(*

short summary
==================
This class tests all methods of xint assertions
with various combinations of inputs and checks expected 
outputs are satisfied or not

.. <legal notes>

legal notes
=================
| SPDX-FileCopyrightText: © 2022 ekvip automation GmbH <info@ekvip.de>
| SPDX-License-Identifier: Apache-2.0
| For details check: Apache-2.0_

.. _Apache-2.0: https://www.apache.org/licenses/LICENSE-2.0

.. </legal notes>

methods and properties
======================

*)

FUNCTION_BLOCK XintAssertionTests EXTENDS AbstractAssertorTest
VAR_INPUT
END_VAR
VAR CONSTANT
	(* prefix to unify the test names *)
	TEST_NAME_PREFIX	:Tc2_System.T_MaxString := 'assert.integer.signed.x.';
	(* number of the lsb *)
	FIRST_BIT				:USINT := 0;
	(* number of the msb *)
	LAST_BIT				:USINT := ((SIZEOF(__XINT)*8)-1);
	(* since we don't know the lenght of __XINT we need it to initialize ``MULTIPLICAND`` *)
	{attribute 'hide'}
	INIT_VALUE_MULTIPLICAND	:__XWORD := 16#1111_1111;
	(* multiplicand for the ``multiplier`` *)
	MULTIPLICAND			:__XINT := (ROR(INIT_VALUE_MULTIPLICAND, 32) OR INIT_VALUE_MULTIPLICAND);
	(* first of all multipliers the test iterates *)
	FIRST_MULTIPLIER		:__XINT := 0;
	(* first of all multipliers the test iterates *)
	LAST_MULTIPLIER			:__XINT := 15;
	(* just the value zero *)
	ZERO					:__XINT := 0;
	(* just the lsb is set, it's just the value one *)
	LSB_ONLY				:__XINT := 1;
	(* all bits are set *)
	ALL_BITS_SET			:__XINT := -1;
	(* the msb is set only *)
	MINIMUM_VALUE			:__XINT := ROR(LSB_ONLY,1);
	(* 
	since we don't know the lenght of __XINT 
	we need it to initialize ``MAXIMUM_VALUE``.
	SHR is not working with __XINT
	*)
	{attribute 'hide'}
	BINARY_MINUS_ONE		:__XWORD := ALL_BITS_SET;
	(* the msb is unset only *)
	MAXIMUM_VALUE			:__XINT := SHR(BINARY_MINUS_ONE,1);
END_VAR

THIS^.runValueIsEqualToTests();
THIS^.runValueIsEvenTests();
THIS^.runValueIsGreaterTests();
THIS^.runValueIsInRangeOfTests();
THIS^.runValueIsLessThanTests();
THIS^.runValueIsMaxTests();
THIS^.runValueIsMinTests();
THIS^.runValueIsNegativeTests();
THIS^.runValueIsNotEqualToTests();
THIS^.runValueIsOddTests();
THIS^.runValueIsPositiveTests();

(*

short summary
==================
This test method is a helper function to create a unified test name

.. <legal notes>

legal notes
=================
| SPDX-FileCopyrightText: © 2022 ekvip automation GmbH <info@ekvip.de>
| SPDX-License-Identifier: Apache-2.0
| For details check: Apache-2.0_

.. _Apache-2.0: https://www.apache.org/licenses/LICENSE-2.0

.. </legal notes>

parameters
==========

*)

METHOD PROTECTED getTestNameFor :Tc2_System.T_MaxString
VAR_INPUT
	(* name of the method to test, to create a unified test name *)
	nameOfMethodToTest	:Tc2_System.T_MaxString;
END_VAR
getTestNameFor := Tc2_Standard.CONCAT(THIS^.TEST_NAME_PREFIX, nameOfMethodToTest);
END_METHOD

(*

short summary
==================
This test method tests ``assert.integer.signed.x.valueIsEqualTo``
method of CNM_AssertionInterfaceLib library with various inputs

.. <legal notes>

legal notes
=================
| SPDX-FileCopyrightText: © 2022 ekvip automation GmbH <info@ekvip.de>
| SPDX-License-Identifier: Apache-2.0
| For details check: Apache-2.0_

.. _Apache-2.0: https://www.apache.org/licenses/LICENSE-2.0

.. </legal notes>

*)

METHOD runValueIsEqualToTests
RETURN (NOT TcUnit.TEST_ORDERED(THIS^.getTestNameFor('valueIsEqualTo')));

THIS^.testValueIsEqualTo(
	valueToTest := THIS^.ZERO,
	expected := THIS^.ALL_BITS_SET
);
THIS^.testValueIsEqualTo(
	valueToTest := THIS^.ZERO,
	expected := THIS^.ZERO
);
THIS^.testValueIsEqualTo(
	valueToTest := THIS^.ALL_BITS_SET,
	expected := THIS^.ALL_BITS_SET
);
THIS^.testValueIsEqualTo(
	valueToTest := THIS^.ALL_BITS_SET,
	expected := THIS^.ZERO
);
THIS^.testValueIsEqualTo(
	valueToTest := THIS^.LSB_ONLY,
	expected := THIS^.LSB_ONLY
);
THIS^.testValueIsEqualTo(
	valueToTest := THIS^.LSB_ONLY,
	expected := THIS^.MINIMUM_VALUE
);
THIS^.testValueIsEqualTo(
	valueToTest := THIS^.MINIMUM_VALUE,
	expected := THIS^.MINIMUM_VALUE
);
THIS^.testValueIsEqualTo(
	valueToTest := THIS^.MINIMUM_VALUE,
	expected := THIS^.LSB_ONLY
);
THIS^.testValueIsEqualTo(
	valueToTest := THIS^.MINIMUM_VALUE,
	expected := THIS^.MAXIMUM_VALUE
);

TcUnit.TEST_FINISHED();
END_METHOD

(*

short summary
==================
This test method tests ``assert.integer.signed.x.valueIsEven``
of CNM_AssertionInterfaceLib library with various inputs

.. <legal notes>

legal notes
=================
| SPDX-FileCopyrightText: © 2022 ekvip automation GmbH <info@ekvip.de>
| SPDX-License-Identifier: Apache-2.0
| For details check: Apache-2.0_

.. _Apache-2.0: https://www.apache.org/licenses/LICENSE-2.0

.. </legal notes>

*)

METHOD runValueIsEvenTests
VAR
	(* it's just part of the test data *)
	valueToTest	:__XINT;
	(* multiplier to get various bit patterns *)
	multiplier	:__XINT;
END_VAR
RETURN (NOT TcUnit.TEST_ORDERED(THIS^.getTestNameFor('valueIsEven')));

FOR multiplier := THIS^.FIRST_MULTIPLIER TO THIS^.LAST_MULTIPLIER DO
	valueToTest := (THIS^.MULTIPLICAND * multiplier);
	THIS^.testValueIsEven(
		valueToTest := valueToTest
	);
END_FOR

TcUnit.TEST_FINISHED();
END_METHOD

(*

short summary
==================
This test method tests ``assert.integer.signed.x.valueIsGreaterThan``
method of CNM_AssertionInterfaceLib library with various inputs

.. <legal notes>

legal notes
=================
| SPDX-FileCopyrightText: © 2022 ekvip automation GmbH <info@ekvip.de>
| SPDX-License-Identifier: Apache-2.0
| For details check: Apache-2.0_

.. _Apache-2.0: https://www.apache.org/licenses/LICENSE-2.0

.. </legal notes>

*)

METHOD runValueIsGreaterTests
RETURN (NOT TcUnit.TEST_ORDERED(THIS^.getTestNameFor('valueIsGreaterThan')));

THIS^.testValueIsGreater(
	valueToTest := THIS^.ZERO,
	less := THIS^.ALL_BITS_SET
);
THIS^.testValueIsGreater(
	valueToTest := THIS^.ZERO,
	less := THIS^.ZERO
);
THIS^.testValueIsGreater(
	valueToTest := THIS^.ALL_BITS_SET,
	less := THIS^.ALL_BITS_SET
);
THIS^.testValueIsGreater(
	valueToTest := THIS^.ALL_BITS_SET,
	less := THIS^.ZERO
);
THIS^.testValueIsGreater(
	valueToTest := THIS^.LSB_ONLY,
	less := THIS^.LSB_ONLY
);
THIS^.testValueIsGreater(
	valueToTest := THIS^.LSB_ONLY,
	less := THIS^.ZERO
);
THIS^.testValueIsGreater(
	valueToTest := THIS^.LSB_ONLY,
	less := (THIS^.LSB_ONLY+THIS^.LSB_ONLY)
);
THIS^.testValueIsGreater(
	valueToTest := THIS^.MINIMUM_VALUE,
	less := THIS^.MINIMUM_VALUE
);
THIS^.testValueIsGreater(
	valueToTest := THIS^.MINIMUM_VALUE,
	less := THIS^.ALL_BITS_SET
);
THIS^.testValueIsGreater(
	valueToTest := THIS^.MINIMUM_VALUE,
	less := THIS^.MAXIMUM_VALUE
);
THIS^.testValueIsGreater(
	valueToTest := THIS^.MAXIMUM_VALUE,
	less := THIS^.MINIMUM_VALUE
);

TcUnit.TEST_FINISHED();
END_METHOD

(*

short summary
==================
This test method tests ``assert.integer.signed.x.valueIsInRangeOf``
method of CNM_AssertionInterfaceLib library with various inputs

.. <legal notes>

legal notes
=================
| SPDX-FileCopyrightText: © 2022 ekvip automation GmbH <info@ekvip.de>
| SPDX-License-Identifier: Apache-2.0
| For details check: Apache-2.0_

.. _Apache-2.0: https://www.apache.org/licenses/LICENSE-2.0

.. </legal notes>

*)

METHOD runValueIsInRangeOfTests
RETURN (NOT TcUnit.TEST_ORDERED(THIS^.getTestNameFor('valueIsInRangeOf')));

THIS^.testValueIsInRangeOf(
	lower := THIS^.ZERO,
	valueToTest := THIS^.LSB_ONLY,
	upper := THIS^.ALL_BITS_SET
);
THIS^.testValueIsInRangeOf(
	lower := THIS^.ZERO,
	valueToTest := THIS^.ZERO,
	upper := THIS^.ZERO
);
THIS^.testValueIsInRangeOf(
	lower := THIS^.ALL_BITS_SET,
	valueToTest := THIS^.ALL_BITS_SET,
	upper := THIS^.ALL_BITS_SET
);
THIS^.testValueIsInRangeOf(
	lower := THIS^.ALL_BITS_SET,
	valueToTest := THIS^.LSB_ONLY,
	upper := THIS^.ZERO
);
THIS^.testValueIsInRangeOf(
	lower := THIS^.ALL_BITS_SET,
	valueToTest := THIS^.ZERO,
	upper := THIS^.ZERO
);
THIS^.testValueIsInRangeOf(
	lower := THIS^.MAXIMUM_VALUE,
	valueToTest := THIS^.ZERO,
	upper := THIS^.MINIMUM_VALUE
);
THIS^.testValueIsInRangeOf(
	lower := THIS^.MINIMUM_VALUE,
	valueToTest := THIS^.ZERO,
	upper := THIS^.MAXIMUM_VALUE
);
THIS^.testValueIsInRangeOf(
	lower := THIS^.MAXIMUM_VALUE,
	valueToTest := THIS^.MINIMUM_VALUE,
	upper := THIS^.MINIMUM_VALUE
);
THIS^.testValueIsInRangeOf(
	lower := THIS^.MINIMUM_VALUE,
	valueToTest := THIS^.MAXIMUM_VALUE,
	upper := THIS^.MAXIMUM_VALUE
);
THIS^.testValueIsInRangeOf(
	lower := THIS^.MINIMUM_VALUE,
	valueToTest := THIS^.MINIMUM_VALUE,
	upper := THIS^.MAXIMUM_VALUE
);

TEST_FINISHED();
END_METHOD

(*

short summary
==================
This test method tests ``assert.integer.signed.x.valueIsLessThan``
method of CNM_AssertionInterfaceLib library with various inputs

.. <legal notes>

legal notes
=================
| SPDX-FileCopyrightText: © 2022 ekvip automation GmbH <info@ekvip.de>
| SPDX-License-Identifier: Apache-2.0
| For details check: Apache-2.0_

.. _Apache-2.0: https://www.apache.org/licenses/LICENSE-2.0

.. </legal notes>

*)

METHOD runValueIsLessThanTests
RETURN (NOT TcUnit.TEST_ORDERED(THIS^.getTestNameFor('valueIsLessThan')));

THIS^.testValueIsLessThan(
	valueToTest := THIS^.ZERO,
	greater := THIS^.ALL_BITS_SET
);
THIS^.testValueIsLessThan(
	valueToTest := THIS^.ZERO,
	greater := THIS^.ZERO
);
THIS^.testValueIsLessThan(
	valueToTest := THIS^.ALL_BITS_SET,
	greater := THIS^.ALL_BITS_SET
);
THIS^.testValueIsLessThan(
	valueToTest := THIS^.ALL_BITS_SET,
	greater := THIS^.ZERO
);
THIS^.testValueIsLessThan(
	valueToTest := THIS^.LSB_ONLY,
	greater := THIS^.LSB_ONLY
);
THIS^.testValueIsLessThan(
	valueToTest := THIS^.LSB_ONLY,
	greater := THIS^.ZERO
);
THIS^.testValueIsLessThan(
	valueToTest := THIS^.MINIMUM_VALUE,
	greater := (THIS^.MINIMUM_VALUE+THIS^.LSB_ONLY)
);
THIS^.testValueIsLessThan(
	valueToTest := THIS^.MINIMUM_VALUE,
	greater := THIS^.MINIMUM_VALUE
);
THIS^.testValueIsLessThan(
	valueToTest := THIS^.MINIMUM_VALUE,
	greater := THIS^.ALL_BITS_SET
);
THIS^.testValueIsLessThan(
	valueToTest := THIS^.MINIMUM_VALUE,
	greater := THIS^.MAXIMUM_VALUE
);
THIS^.testValueIsLessThan(
	valueToTest := THIS^.MAXIMUM_VALUE,
	greater := THIS^.MINIMUM_VALUE
);

TcUnit.TEST_FINISHED();
END_METHOD

(*

short summary
==================
This test method tests ``assert.integer.signed.x.valueIsMax``
method of CNM_AssertionInterfaceLib library with various inputs

.. <legal notes>

legal notes
=================
| SPDX-FileCopyrightText: © 2022 ekvip automation GmbH <info@ekvip.de>
| SPDX-License-Identifier: Apache-2.0
| For details check: Apache-2.0_

.. _Apache-2.0: https://www.apache.org/licenses/LICENSE-2.0

.. </legal notes>

*)

METHOD runValueIsMaxTests
RETURN (NOT TcUnit.TEST_ORDERED(THIS^.getTestNameFor('valueIsMax')));

THIS^.testValueIsMax(
	valueToTest := THIS^.ZERO,
	maximum := THIS^.LSB_ONLY
);
THIS^.testValueIsMax(
	valueToTest := THIS^.LSB_ONLY,
	maximum := THIS^.ZERO
);
THIS^.testValueIsMax(
	valueToTest := THIS^.ZERO,
	maximum := THIS^.ZERO
);
THIS^.testValueIsMax(
	valueToTest := THIS^.ALL_BITS_SET,
	maximum := ALL_BITS_SET
);
THIS^.testValueIsMax(
	valueToTest := (THIS^.ALL_BITS_SET-THIS^.LSB_ONLY),
	maximum := THIS^.ALL_BITS_SET
);
THIS^.testValueIsMax(
	valueToTest := THIS^.ALL_BITS_SET,
	maximum := (THIS^.ALL_BITS_SET-THIS^.LSB_ONLY)
);
THIS^.testValueIsMax(
	valueToTest := THIS^.MINIMUM_VALUE,
	maximum := (THIS^.MINIMUM_VALUE+THIS^.LSB_ONLY)
);
THIS^.testValueIsMax(
	valueToTest := (THIS^.MINIMUM_VALUE+THIS^.LSB_ONLY),
	maximum := THIS^.MINIMUM_VALUE
);
THIS^.testValueIsMax(
	valueToTest := THIS^.MINIMUM_VALUE,
	maximum := THIS^.MINIMUM_VALUE
);
THIS^.testValueIsMax(
	valueToTest := THIS^.MINIMUM_VALUE,
	maximum := THIS^.MAXIMUM_VALUE
);
THIS^.testValueIsMax(
	valueToTest := THIS^.MAXIMUM_VALUE,
	maximum := THIS^.MINIMUM_VALUE
);

TcUnit.TEST_FINISHED();
END_METHOD

(*

short summary
==================
This test method tests ``assert.integer.signed.x.valueIsMin``
method of CNM_AssertionInterfaceLib library with various inputs

.. <legal notes>

legal notes
=================
| SPDX-FileCopyrightText: © 2022 ekvip automation GmbH <info@ekvip.de>
| SPDX-License-Identifier: Apache-2.0
| For details check: Apache-2.0_

.. _Apache-2.0: https://www.apache.org/licenses/LICENSE-2.0

.. </legal notes>

*)

METHOD runValueIsMinTests
RETURN (NOT TcUnit.TEST_ORDERED(THIS^.getTestNameFor('valueIsMin')));

THIS^.testValueIsMin(
	valueToTest := THIS^.ZERO,
	minimum := THIS^.LSB_ONLY
);
THIS^.testValueIsMin(
	valueToTest := THIS^.LSB_ONLY,
	minimum := THIS^.ZERO
);
THIS^.testValueIsMin(
	valueToTest := THIS^.ZERO,
	minimum := THIS^.ZERO
);
THIS^.testValueIsMin(
	valueToTest := THIS^.ALL_BITS_SET,
	minimum := ALL_BITS_SET
);
THIS^.testValueIsMin(
	valueToTest := (THIS^.ALL_BITS_SET-THIS^.LSB_ONLY),
	minimum := THIS^.ALL_BITS_SET
);
THIS^.testValueIsMin(
	valueToTest := THIS^.ALL_BITS_SET,
	minimum := (THIS^.ALL_BITS_SET-THIS^.LSB_ONLY)
);
THIS^.testValueIsMin(
	valueToTest := THIS^.MINIMUM_VALUE,
	minimum := (THIS^.MINIMUM_VALUE+THIS^.LSB_ONLY)
);
THIS^.testValueIsMin(
	valueToTest := (THIS^.MINIMUM_VALUE+THIS^.LSB_ONLY),
	minimum := THIS^.MINIMUM_VALUE
);
THIS^.testValueIsMin(
	valueToTest := THIS^.MINIMUM_VALUE,
	minimum := THIS^.MINIMUM_VALUE
);
THIS^.testValueIsMin(
	valueToTest := THIS^.MINIMUM_VALUE,
	minimum := THIS^.MAXIMUM_VALUE
);
THIS^.testValueIsMin(
	valueToTest := THIS^.MAXIMUM_VALUE,
	minimum := THIS^.MINIMUM_VALUE
);

TcUnit.TEST_FINISHED();
END_METHOD

(*

short summary
==================
This test method tests ``assert.integer.signed.x.valueIsNegative``
of CNM_AssertionInterfaceLib library with various inputs

.. <legal notes>

legal notes
=================
| SPDX-FileCopyrightText: © 2022 ekvip automation GmbH <info@ekvip.de>
| SPDX-License-Identifier: Apache-2.0
| For details check: Apache-2.0_

.. _Apache-2.0: https://www.apache.org/licenses/LICENSE-2.0

.. </legal notes>

*)

METHOD runValueIsNegativeTests
VAR
	(* it's just part of the test data *)
	valueToTest	:__XINT;
	(* multiplier to get various bit patterns *)
	multiplier	:__XINT;
END_VAR
RETURN (NOT TcUnit.TEST_ORDERED(THIS^.getTestNameFor('valueIsNegative')));

FOR multiplier := THIS^.FIRST_MULTIPLIER TO THIS^.LAST_MULTIPLIER DO
	valueToTest := (THIS^.MULTIPLICAND * multiplier);
	THIS^.testValueIsNegative(
		valueToTest := valueToTest
	);
END_FOR

TcUnit.TEST_FINISHED();
END_METHOD

(*

short summary
==================
This test method tests ``assert.integer.signed.x.valueIsNotEqualTo``
method of CNM_AssertionInterfaceLib library with various inputs

.. <legal notes>

legal notes
=================
| SPDX-FileCopyrightText: © 2022 ekvip automation GmbH <info@ekvip.de>
| SPDX-License-Identifier: Apache-2.0
| For details check: Apache-2.0_

.. _Apache-2.0: https://www.apache.org/licenses/LICENSE-2.0

.. </legal notes>

*)

METHOD runValueIsNotEqualToTests
RETURN (NOT TcUnit.TEST_ORDERED(THIS^.getTestNameFor('valueIsNotEqualTo')));

THIS^.testValueIsNotEqualTo(
	valueToTest := THIS^.ZERO,
	unexpected := THIS^.ALL_BITS_SET
);
THIS^.testValueIsNotEqualTo(
	valueToTest := THIS^.ZERO,
	unexpected := THIS^.ZERO
);
THIS^.testValueIsNotEqualTo(
	valueToTest := THIS^.ALL_BITS_SET,
	unexpected := THIS^.ALL_BITS_SET
);
THIS^.testValueIsNotEqualTo(
	valueToTest := THIS^.ALL_BITS_SET,
	unexpected := THIS^.ZERO
);
THIS^.testValueIsNotEqualTo(
	valueToTest := THIS^.LSB_ONLY,
	unexpected := THIS^.LSB_ONLY
);
THIS^.testValueIsNotEqualTo(
	valueToTest := THIS^.LSB_ONLY,
	unexpected := THIS^.MINIMUM_VALUE
);
THIS^.testValueIsNotEqualTo(
	valueToTest := THIS^.MINIMUM_VALUE,
	unexpected := THIS^.MINIMUM_VALUE
);
THIS^.testValueIsNotEqualTo(
	valueToTest := THIS^.MINIMUM_VALUE,
	unexpected := THIS^.LSB_ONLY
);
THIS^.testValueIsNotEqualTo(
	valueToTest := THIS^.MINIMUM_VALUE,
	unexpected := THIS^.MAXIMUM_VALUE
);

TcUnit.TEST_FINISHED();
END_METHOD

(*

short summary
==================
This test method tests ``assert.integer.signed.x.valueIsOdd``
of CNM_AssertionInterfaceLib library with various inputs

.. <legal notes>

legal notes
=================
| SPDX-FileCopyrightText: © 2022 ekvip automation GmbH <info@ekvip.de>
| SPDX-License-Identifier: Apache-2.0
| For details check: Apache-2.0_

.. _Apache-2.0: https://www.apache.org/licenses/LICENSE-2.0

.. </legal notes>

*)

METHOD runValueIsOddTests
VAR
	(* it's just part of the test data *)
	valueToTest	:__XINT;
	(* multiplier to get various bit patterns *)
	multiplier	:__XINT;
END_VAR
RETURN (NOT TcUnit.TEST_ORDERED(THIS^.getTestNameFor('valueIsOdd')));

FOR multiplier := THIS^.FIRST_MULTIPLIER TO THIS^.LAST_MULTIPLIER DO
	valueToTest := (THIS^.MULTIPLICAND * multiplier);
	THIS^.testValueIsOdd(
		valueToTest := valueToTest
	);
END_FOR

TcUnit.TEST_FINISHED();
END_METHOD

(*

short summary
==================
This test method tests ``assert.integer.signed.x.valueIsPositive``
of CNM_AssertionInterfaceLib library with various inputs

.. <legal notes>

legal notes
=================
| SPDX-FileCopyrightText: © 2022 ekvip automation GmbH <info@ekvip.de>
| SPDX-License-Identifier: Apache-2.0
| For details check: Apache-2.0_

.. _Apache-2.0: https://www.apache.org/licenses/LICENSE-2.0

.. </legal notes>

*)

METHOD runValueIsPositiveTests
VAR
	(* it's just part of the test data *)
	valueToTest	:__XINT;
	(* multiplier to get various bit patterns *)
	multiplier	:__XINT;
END_VAR
RETURN (NOT TcUnit.TEST_ORDERED(THIS^.getTestNameFor('valueIsPositive')));

FOR multiplier := THIS^.FIRST_MULTIPLIER TO THIS^.LAST_MULTIPLIER DO
	valueToTest := (THIS^.MULTIPLICAND * multiplier);
	THIS^.testValueIsPositive(
		valueToTest := valueToTest
	);
END_FOR

TcUnit.TEST_FINISHED();
END_METHOD

(*

short summary
==================
This test method tests ``assert.integer.signed.x.valueIsEqualTo``
method of CNM_AssertionInterfaceLib library, 
it provides the possibility to handover test data via parameter 


.. <legal notes>

legal notes
=================
| SPDX-FileCopyrightText: © 2022 ekvip automation GmbH <info@ekvip.de>
| SPDX-License-Identifier: Apache-2.0
| For details check: Apache-2.0_

.. _Apache-2.0: https://www.apache.org/licenses/LICENSE-2.0

.. </legal notes>

parameters
==========

*)

METHOD testValueIsEqualTo
VAR_INPUT
	(* for the test it's the parameter ``currentValue`` *)
	valueToTest	:__XINT;
	(* for the test it's the parameter ``expectedValue`` *)
	expected	:__XINT;
END_VAR
VAR
	(* just the expectation if the assertion to test must be worng or true *)
	assertionIsWrong		:BOOL;
	(* contains the format string for the test message *)
	message					:Tc2_System.T_MaxString;
	(* TwinCAT printf with the test message *)
	messageStringBuilder	:Tc2_Utilities.FB_FormatString;
END_VAR
THIS^.assertorContainer.resetAssertor();

assertionIsWrong := (valueToTest <> expected);
message := SEL(
	assertionIsWrong,
	'currentValue is %d expectedValue is %d assertion must be TRUE', 
	'currentValue is %d expectedValue is %d assertion must be FALSE'
);
messageStringBuilder(
	sFormat := message,
	arg1 := THIS^.AnyToArg(valueToTest),
	arg2 := THIS^.AnyToArg(expected)
);

THIS^.assertorContainer.assertor.assert.integer.signed.x.valueIsEqualTo(
	currentValue := valueToTest,
	expectedValue := expected,
	message := ''
);

THIS^.AssertEquals_BOOL(
	Expected 	:= assertionIsWrong,
	Actual 		:= THIS^.assertorContainer.wasAssertionWrong,
	Message 	:= messageStringBuilder.sOut
);
END_METHOD

(*

short summary
==================
This test method tests ``assert.integer.signed.x.valueIsEven``
of CNM_AssertionInterfaceLib library, 
it provides the possibility to handover test data via parameter 


.. <legal notes>

legal notes
=================
| SPDX-FileCopyrightText: © 2022 ekvip automation GmbH <info@ekvip.de>
| SPDX-License-Identifier: Apache-2.0
| For details check: Apache-2.0_

.. _Apache-2.0: https://www.apache.org/licenses/LICENSE-2.0

.. </legal notes>

parameters
==========

*)

METHOD testValueIsEven
VAR_INPUT
	(* for the test it's the parameter ``currentValue`` *)
	valueToTest	:__XINT;
END_VAR
VAR
	(* just the expectation if the assertion to test must be worng or true *)
	assertionIsWrong		:BOOL;
	(* contains the format string for the test message *)
	message					:Tc2_System.T_MaxString;
	(* TwinCAT printf with the test message *)
	messageStringBuilder	:Tc2_Utilities.FB_FormatString;
END_VAR
THIS^.assertorContainer.resetAssertor();

assertionIsWrong := (valueToTest.FIRST_BIT);

message := SEL(
	assertionIsWrong,
	'currentValue is %d assertion must be TRUE',
	'currentValue is %d assertion must be FALSE'
);

messageStringBuilder(
	sFormat := message,
	arg1 := THIS^.AnyToArg(valueToTest)
);

THIS^.assertorContainer.assertor.assert.integer.signed.x.valueIsEven(
	currentValue 	:= valueToTest,
	message			:= ''  
); 

THIS^.AssertEquals_BOOL(
	Expected 	:= assertionIsWrong,
	Actual 		:= THIS^.assertorContainer.wasAssertionWrong,
	Message 	:= messageStringBuilder.sOut
);
END_METHOD

(*

short summary
==================
This test method tests ``assert.integer.signed.x.valueIsGreaterThan``
method of CNM_AssertionInterfaceLib library, 
it provides the possibility to handover test data via parameter 


.. <legal notes>

legal notes
=================
| SPDX-FileCopyrightText: © 2022 ekvip automation GmbH <info@ekvip.de>
| SPDX-License-Identifier: Apache-2.0
| For details check: Apache-2.0_

.. _Apache-2.0: https://www.apache.org/licenses/LICENSE-2.0

.. </legal notes>

parameters
==========

*)

METHOD testValueIsGreater
VAR_INPUT
	(* for the test it's the parameter ``currentValue`` *)
	valueToTest	:__XINT;
	(* for the test it's the parameter ``lessValue`` *)
	less		:__XINT;
END_VAR
VAR
	(* just the expectation if the assertion to test must be worng or true *)
	assertionIsWrong		:BOOL;
	(* contains the format string for the test message *)
	message					:Tc2_System.T_MaxString;
	(* TwinCAT printf with the test message *)
	messageStringBuilder	:Tc2_Utilities.FB_FormatString;
END_VAR
THIS^.assertorContainer.resetAssertor();

assertionIsWrong := (valueToTest <= less);
message := SEL(
	assertionIsWrong,
	'currentValue is %d lessValue is %d assertion must be TRUE', 
	'currentValue is %d lessValue is %d assertion must be FALSE'
);
messageStringBuilder(
	sFormat := message,
	arg1 := THIS^.AnyToArg(valueToTest),
	arg2 := THIS^.AnyToArg(less)
);

THIS^.assertorContainer.assertor.assert.integer.signed.x.valueIsGreaterThan(
	currentValue := valueToTest,
	lessValue := less,
	message := ''
);

THIS^.AssertEquals_BOOL(
	Expected 	:= assertionIsWrong,
	Actual 		:= THIS^.assertorContainer.wasAssertionWrong,
	Message 	:= messageStringBuilder.sOut
);
END_METHOD

(*

short summary
==================
This test method tests ``assert.integer.signed.x.valueIsInRangeOf``
method of CNM_AssertionInterfaceLib library, 
it provides the possibility to handover test data via parameter 


.. <legal notes>

legal notes
=================
| SPDX-FileCopyrightText: © 2022 ekvip automation GmbH <info@ekvip.de>
| SPDX-License-Identifier: Apache-2.0
| For details check: Apache-2.0_

.. _Apache-2.0: https://www.apache.org/licenses/LICENSE-2.0

.. </legal notes>

parameters
==========

*)

METHOD testValueIsInRangeOf
VAR_INPUT
	(* for the test it's the parameter ``lowerLimit`` *)
	lower		:__XINT;
	(* for the test it's the parameter ``currentValue`` *)
	valueToTest	:__XINT;
	(* for the test it's the parameter ``upperLimit`` *)
	upper		:__XINT;
END_VAR          
VAR
	(* just the expectation if the assertion to test must be worng or true *)
	assertionIsWrong		:BOOL;
	(* contains the format string for the test message *)
	message					:Tc2_System.T_MaxString;
	(* TwinCAT printf with the test message *)
	messageStringBuilder	:Tc2_Utilities.FB_FormatString;
END_VAR
THIS^.assertorContainer.resetAssertor();

assertionIsWrong := ((valueToTest < lower) OR (valueToTest > upper)); 

message := SEL(
	assertionIsWrong,
	'lowerLimit is %d currentValue is %d upperLimit is %d assertion must be TRUE', 
	'lowerLimit is %d currentValue is %d upperLimit is %d assertion must be FALSE'
);

messageStringBuilder(
	sFormat := message,
	arg1 := THIS^.AnyToArg(lower),
	arg2 := THIS^.AnyToArg(valueToTest),
	arg3 := THIS^.AnyToArg(upper)
);

THIS^.assertorContainer.assertor.assert.integer.signed.x.valueIsInRangeOf(
	lowerLimit := lower,
	currentValue := valueToTest,
	upperLimit := upper,
	message := ''
);

THIS^.AssertEquals_BOOL(
	Expected 	:= assertionIsWrong,
	Actual 		:= THIS^.assertorContainer.wasAssertionWrong,
	Message 	:= messageStringBuilder.sOut
);
END_METHOD

(*

short summary
==================
This test method tests ``assert.integer.signed.x.valueIsLessThan``
method of CNM_AssertionInterfaceLib library, 
it provides the possibility to handover test data via parameter 


.. <legal notes>

legal notes
=================
| SPDX-FileCopyrightText: © 2022 ekvip automation GmbH <info@ekvip.de>
| SPDX-License-Identifier: Apache-2.0
| For details check: Apache-2.0_

.. _Apache-2.0: https://www.apache.org/licenses/LICENSE-2.0

.. </legal notes>

parameters
==========

*)

METHOD testValueIsLessThan
VAR_INPUT
	(* for the test it's the parameter ``currentValue`` *)
	valueToTest	:__XINT;
	(* for the test it's the parameter ``greaterValue`` *)
	greater		:__XINT;
END_VAR
VAR
	(* just the expectation if the assertion to test must be worng or true *)
	assertionIsWrong		:BOOL;
	(* contains the format string for the test message *)
	message					:Tc2_System.T_MaxString;
	(* TwinCAT printf with the test message *)
	messageStringBuilder	:Tc2_Utilities.FB_FormatString;
END_VAR
THIS^.assertorContainer.resetAssertor();

assertionIsWrong := (valueToTest >= greater);
message := SEL(
	assertionIsWrong,
	'currentValue is %d greaterValue is %d assertion must be TRUE',
	'currentValue is %d greaterValue is %d assertion must be FALSE'
);
messageStringBuilder(
	sFormat := message,
	arg1 := THIS^.AnyToArg(valueToTest),
	arg2 := THIS^.AnyToArg(greater)
);

THIS^.assertorContainer.assertor.assert.integer.signed.x.valueIsLessThan(
	currentValue := valueToTest,
	greaterValue := greater,
	message := ''
);

THIS^.AssertEquals_BOOL(
	Expected 	:= assertionIsWrong,
	Actual 		:= THIS^.assertorContainer.wasAssertionWrong,
	Message 	:= messageStringBuilder.sOut
);
END_METHOD

(*

short summary
==================
This test method tests ``assert.integer.signed.x.valueIsMax``
method of CNM_AssertionInterfaceLib library, 
it provides the possibility to handover test data via parameter 


.. <legal notes>

legal notes
=================
| SPDX-FileCopyrightText: © 2022 ekvip automation GmbH <info@ekvip.de>
| SPDX-License-Identifier: Apache-2.0
| For details check: Apache-2.0_

.. _Apache-2.0: https://www.apache.org/licenses/LICENSE-2.0

.. </legal notes>

parameters
==========

*)

METHOD testValueIsMax 
VAR_INPUT
	(* for the test it's the parameter ``currentValue`` *)
	valueToTest	:__XINT;
	(* for the test it's the parameter ``maximumValue`` *)
	maximum		:__XINT;
END_VAR
VAR
	(* just the expectation if the assertion to test must be worng or true *)
	assertionIsWrong		:BOOL;
	(* contains the format string for the test message *)
	message					:Tc2_System.T_MaxString;
	(* TwinCAT printf with the test message *)
	messageStringBuilder	:Tc2_Utilities.FB_FormatString;
END_VAR
THIS^.assertorContainer.resetAssertor();

assertionIsWrong := (valueToTest > maximum);
message := SEL(
	assertionIsWrong,
	'currentValue is %d maximumValue is %d assertion must be TRUE',
	'currentValue is %d maximumValue is %d assertion must be FALSE'
);
messageStringBuilder(
	sFormat := message,
	arg1 := THIS^.AnyToArg(valueToTest),
	arg2 := THIS^.AnyToArg(maximum)
);

THIS^.assertorContainer.assertor.assert.integer.signed.x.valueIsMax(
	currentValue := valueToTest,
	maximumValue := maximum,
	message := ''
);

THIS^.AssertEquals_BOOL(
	Expected 	:= assertionIsWrong,
	Actual 		:= THIS^.assertorContainer.wasAssertionWrong,
	Message 	:= messageStringBuilder.sOut
);
END_METHOD

(*

short summary
==================
This test method tests ``assert.integer.signed.x.valueIsMin``
method of CNM_AssertionInterfaceLib library, 
it provides the possibility to handover test data via parameter 


.. <legal notes>

legal notes
=================
| SPDX-FileCopyrightText: © 2022 ekvip automation GmbH <info@ekvip.de>
| SPDX-License-Identifier: Apache-2.0
| For details check: Apache-2.0_

.. _Apache-2.0: https://www.apache.org/licenses/LICENSE-2.0

.. </legal notes>

parameters
==========

*)

METHOD testValueIsMin 
VAR_INPUT
	(* for the test it's the parameter ``currentValue`` *)
	valueToTest	:__XINT;
	(* for the test it's the parameter ``minimumValue`` *)
	minimum		:__XINT;
END_VAR
VAR
	(* just the expectation if the assertion to test must be worng or true *)
	assertionIsWrong		:BOOL;
	(* contains the format string for the test message *)
	message					:Tc2_System.T_MaxString;
	(* TwinCAT printf with the test message *)
	messageStringBuilder	:Tc2_Utilities.FB_FormatString;
END_VAR
THIS^.assertorContainer.resetAssertor();

assertionIsWrong := (valueToTest < minimum);
message := SEL(
	assertionIsWrong,
	'currentValue is %d minimumValue is %d assertion must be TRUE',
	'currentValue is %d minimumValue is %d assertion must be FALSE'
);
messageStringBuilder(
	sFormat := message,
	arg1 := THIS^.AnyToArg(valueToTest),
	arg2 := THIS^.AnyToArg(minimum)
);

THIS^.assertorContainer.assertor.assert.integer.signed.x.valueIsMin(
	currentValue := valueToTest,
	minimumValue := minimum,
	message := ''
);

THIS^.AssertEquals_BOOL(
	Expected 	:= assertionIsWrong,
	Actual 		:= THIS^.assertorContainer.wasAssertionWrong,
	Message 	:= messageStringBuilder.sOut
);
END_METHOD

(*

short summary
==================
This test method tests ``assert.integer.signed.x.valueIsNegative``
of CNM_AssertionInterfaceLib library, 
it provides the possibility to handover test data via parameter 


.. <legal notes>

legal notes
=================
| SPDX-FileCopyrightText: © 2022 ekvip automation GmbH <info@ekvip.de>
| SPDX-License-Identifier: Apache-2.0
| For details check: Apache-2.0_

.. _Apache-2.0: https://www.apache.org/licenses/LICENSE-2.0

.. </legal notes>

parameters
==========

*)

METHOD testValueIsNegative
VAR_INPUT
	(* for the test it's the parameter ``currentValue`` *)
	valueToTest	:__XINT;
END_VAR
VAR
	(* just the expectation if the assertion to test must be worng or true *)
	assertionIsWrong		:BOOL;
	(* contains the format string for the test message *)
	message					:Tc2_System.T_MaxString;
	(* TwinCAT printf with the test message *)
	messageStringBuilder	:Tc2_Utilities.FB_FormatString;
END_VAR
THIS^.assertorContainer.resetAssertor();

assertionIsWrong := (valueToTest >= THIS^.ZERO);

message := SEL(
	assertionIsWrong,
	'currentValue is %d assertion must be TRUE',
	'currentValue is %d assertion must be FALSE'
);

messageStringBuilder(
	sFormat := message,
	arg1 := THIS^.AnyToArg(valueToTest)
);

THIS^.assertorContainer.assertor.assert.integer.signed.x.valueIsNegative(
	currentValue 	:= valueToTest,
	message			:= ''  
); 

THIS^.AssertEquals_BOOL(
	Expected 	:= assertionIsWrong,
	Actual 		:= THIS^.assertorContainer.wasAssertionWrong,
	Message 	:= messageStringBuilder.sOut
);
END_METHOD

(*

short summary
==================
This test method tests ``assert.integer.signed.x.valueIsNotEqualTo``
method of CNM_AssertionInterfaceLib library, 
it provides the possibility to handover test data via parameter 


.. <legal notes>

legal notes
=================
| SPDX-FileCopyrightText: © 2022 ekvip automation GmbH <info@ekvip.de>
| SPDX-License-Identifier: Apache-2.0
| For details check: Apache-2.0_

.. _Apache-2.0: https://www.apache.org/licenses/LICENSE-2.0

.. </legal notes>

parameters
==========

*)

METHOD testValueIsNotEqualTo
VAR_INPUT
	(* for the test it's the parameter ``currentValue`` *)
	valueToTest	:__XINT;
	(* for the test it's the parameter ``unexpectedValue`` *)
	unexpected	:__XINT;
END_VAR
VAR
	(* just the expectation if the assertion to test must be worng or true *)
	assertionIsWrong		:BOOL;
	(* contains the format string for the test message *)
	message					:Tc2_System.T_MaxString;
	(* TwinCAT printf with the test message *)
	messageStringBuilder	:Tc2_Utilities.FB_FormatString;
END_VAR
THIS^.assertorContainer.resetAssertor();

assertionIsWrong := (valueToTest = unexpected);
message := SEL(
	assertionIsWrong,
	'currentValue is %d unexpectedValue is %d assertion must be TRUE', 
	'currentValue is %d unexpectedValue is %d assertion must be FALSE'
);
messageStringBuilder(
	sFormat := message,
	arg1 := THIS^.AnyToArg(valueToTest),
	arg2 := THIS^.AnyToArg(unexpected)
);

THIS^.assertorContainer.assertor.assert.integer.signed.x.valueIsNotEqualTo(
	currentValue := valueToTest,
	unexpectedValue := unexpected,
	message := ''
);

THIS^.AssertEquals_BOOL(
	Expected 	:= assertionIsWrong,
	Actual 		:= THIS^.assertorContainer.wasAssertionWrong,
	Message 	:= messageStringBuilder.sOut
);
END_METHOD

(*

short summary
==================
This test method tests ``assert.integer.signed.x.valueIsOdd``
of CNM_AssertionInterfaceLib library, 
it provides the possibility to handover test data via parameter 


.. <legal notes>

legal notes
=================
| SPDX-FileCopyrightText: © 2022 ekvip automation GmbH <info@ekvip.de>
| SPDX-License-Identifier: Apache-2.0
| For details check: Apache-2.0_

.. _Apache-2.0: https://www.apache.org/licenses/LICENSE-2.0

.. </legal notes>

parameters
==========

*)

METHOD testValueIsOdd
VAR_INPUT
	(* for the test it's the parameter ``currentValue`` *)
	valueToTest	:__XINT;
END_VAR
VAR
	(* just the expectation if the assertion to test must be worng or true *)
	assertionIsWrong		:BOOL;
	(* contains the format string for the test message *)
	message					:Tc2_System.T_MaxString;
	(* TwinCAT printf with the test message *)
	messageStringBuilder	:Tc2_Utilities.FB_FormatString;
END_VAR
THIS^.assertorContainer.resetAssertor();

assertionIsWrong := (NOT valueToTest.FIRST_BIT);

message := SEL(
	assertionIsWrong,
	'currentValue is %d assertion must be TRUE',
	'currentValue is %d assertion must be FALSE'
);

messageStringBuilder(
	sFormat := message,
	arg1 := THIS^.AnyToArg(valueToTest)
);

THIS^.assertorContainer.assertor.assert.integer.signed.x.valueIsOdd(
	currentValue 	:= valueToTest,
	message			:= ''  
); 

THIS^.AssertEquals_BOOL(
	Expected 	:= assertionIsWrong,
	Actual 		:= THIS^.assertorContainer.wasAssertionWrong,
	Message 	:= messageStringBuilder.sOut
);
END_METHOD

(*

short summary
==================
This test method tests ``assert.integer.signed.x.valueIsPositive``
of CNM_AssertionInterfaceLib library, 
it provides the possibility to handover test data via parameter 


.. <legal notes>

legal notes
=================
| SPDX-FileCopyrightText: © 2022 ekvip automation GmbH <info@ekvip.de>
| SPDX-License-Identifier: Apache-2.0
| For details check: Apache-2.0_

.. _Apache-2.0: https://www.apache.org/licenses/LICENSE-2.0

.. </legal notes>

parameters
==========

*)

METHOD testValueIsPositive
VAR_INPUT
	(* for the test it's the parameter ``currentValue`` *)
	valueToTest	:__XINT;
END_VAR
VAR
	(* just the expectation if the assertion to test must be worng or true *)
	assertionIsWrong		:BOOL;
	(* contains the format string for the test message *)
	message					:Tc2_System.T_MaxString;
	(* TwinCAT printf with the test message *)
	messageStringBuilder	:Tc2_Utilities.FB_FormatString;
END_VAR
THIS^.assertorContainer.resetAssertor();

assertionIsWrong := (valueToTest < THIS^.ZERO);

message := SEL(
	assertionIsWrong,
	'currentValue is %d assertion must be TRUE',
	'currentValue is %d assertion must be FALSE'
);

messageStringBuilder(
	sFormat := message,
	arg1 := THIS^.AnyToArg(valueToTest)
);

THIS^.assertorContainer.assertor.assert.integer.signed.x.valueIsPositive(
	currentValue 	:= valueToTest,
	message			:= ''  
); 

THIS^.AssertEquals_BOOL(
	Expected 	:= assertionIsWrong,
	Actual 		:= THIS^.assertorContainer.wasAssertionWrong,
	Message 	:= messageStringBuilder.sOut
);
END_METHOD

END_FUNCTION_BLOCK

(* stored: Version 1.1.0.1, ProductVersion 3.1.4024.12
   POU XintAssertionTests: Id {a1e1e542-9410-478f-9227-7f03178f770e}, SpecialFunc None
   Folder internal: Id {84422967-87ac-41d2-829d-147352469888}
   Folder valueIsEqualTo: Id {b697e7e3-2828-41a1-b0d6-a3a1a7708beb}
   Folder valueIsEven: Id {4e23cc7b-5254-43b4-9b85-6a0f48deae57}
   Folder valueIsGreaterThan: Id {09c5b36d-9457-43b1-8c97-dac188123443}
   Folder valueIsInRangeOf: Id {314e71a4-df67-4159-bd6d-e11c060bf47d}
   Folder valueIsLessThan: Id {42fc5448-d177-4cec-bf32-8b58d3a3b627}
   Folder valueIsMax: Id {66be3a5c-5492-46c5-8c3d-1b2e33c14a11}
   Folder valueIsMin: Id {e9495d21-cb11-4b4a-b6e6-5b07b3efb788}
   Folder valueIsNegative: Id {e1b19ea8-48f5-4e6c-9d54-b8534edcb5ca}
   Folder valueIsNotEqual: Id {06666869-b91e-420e-b884-f61074450902}
   Folder valueIsOdd: Id {5edb1a27-19ae-44b3-8fb8-57f802d5a5cf}
   Folder valueIsPositive: Id {3e51f832-bbc5-4d13-ae32-d9b9d17993d8}
   Method getTestNameFor: Id {51394b35-db0d-4457-a1a6-59c5d2552e4e}
   Method runValueIsEqualToTests: Id {2c6b40b1-6c65-453d-bc34-fbf5d2d84918}
   Method runValueIsEvenTests: Id {79db37d9-a1b6-4c78-884f-471b38dcfb11}
   Method runValueIsGreaterTests: Id {b06f7919-3766-4b7e-a0f6-f9cb78e61d0d}
   Method runValueIsInRangeOfTests: Id {040c47ae-9cef-4644-8d5f-a4c442c2d56a}
   Method runValueIsLessThanTests: Id {e115664b-5eea-402f-96e0-9b46ae342992}
   Method runValueIsMaxTests: Id {737c1fcf-71fc-45fe-ac93-fdae53323670}
   Method runValueIsMinTests: Id {19a5917d-b3d6-492e-a56f-02af1afe5a0b}
   Method runValueIsNegativeTests: Id {3b4c9b72-9559-4da6-ab02-6b04b6c5fed6}
   Method runValueIsNotEqualToTests: Id {371fe5cb-a338-45c1-b7db-673c4cb594fc}
   Method runValueIsOddTests: Id {8e6e5f26-778a-4b74-9b5a-498778e01eb1}
   Method runValueIsPositiveTests: Id {cc17bead-3825-4a84-9c00-75cf22c14fb2}
   Method testValueIsEqualTo: Id {efcb47e5-e57a-49f4-bcd7-c291c3871d7a}
   Method testValueIsEven: Id {d3bf9041-415d-41c8-8d9f-104c7fd8ab94}
   Method testValueIsGreater: Id {71880131-9865-47f6-9f4d-98d5b9fdd3c5}
   Method testValueIsInRangeOf: Id {2f5ae3ca-addf-47b2-91c3-94a9658d458b}
   Method testValueIsLessThan: Id {0b1a2a36-3be6-452e-a3db-5d4d53ef5a73}
   Method testValueIsMax: Id {69f014fc-08e2-405b-b1ce-76e754f62569}
   Method testValueIsMin: Id {a173638d-3db0-4e8f-9bc1-0192480e2062}
   Method testValueIsNegative: Id {5e2a5f67-80cb-464f-a704-e195dd36af20}
   Method testValueIsNotEqualTo: Id {80707e5a-5583-4e3a-bea7-344595c1b894}
   Method testValueIsOdd: Id {b50ef440-eefd-4cd7-a0e4-2aebd27c4eca}
   Method testValueIsPositive: Id {9dd84e3e-6165-4982-8e93-9b110dd749bf} *)
